// Implicitly generated code : DO NOT EDIT
FUNCTION CheckDivDInt : DINT
VAR_INPUT
	divisor:DINT;
END_VAR

// Implicitly generated code : Only an Implementation suggestion
{noflow}
IF divisor = 0 THEN
	CheckDivDInt:=1;
ELSE
	CheckDivDInt:=divisor;
END_IF;
{flow}

END_FUNCTION

(* stored: Version 1.1.0.1, ProductVersion 3.1.4024.11
   POU CheckDivDInt: Id {54154234-9f9b-0574-1bce-485238e579c3}, SpecialFunc CheckDivInt32 *)
